// TIA Portal V20 export
TYPE "LCFL_typeMTPMonBinVlv"
TITLE = MTP for monitoring binary valve / MTP für binäre Ventilüberwachung
// MTP data for bistable valve with the feedback monitoring / MTP-Daten für bistabiles Ventil mit Rückmeldeüberwachung
   STRUCT
      WQC { ExternalWritable := 'False'} : Byte := 16#FF;   // Schlechtester Quality Code / Worst quality code
      OSLevel : Byte := 16#00;   // OS-Level / OS level
      StateChannel { ExternalWritable := 'False'} : Bool := FALSE;   // Auswahl des aktiven Betriebsart-Interaktionskanals (0: Die Bedienschalter (*Op) sind zu verwenden; 1: Die automatischen Schalter (*Aut) sind zu verwenden) / Selection of the active operation mode interaction channel (0: The operator switches (*Op) shall be used; 1: The automatic switches (*Aut) shall be used)
      StateOffAut { ExternalWritable := 'False'} : Bool := FALSE;   // Betriebsart durch automatische Interaktion auf "Aus" setzen (relevant, wenn StateChannel = 1) (1: Betriebsart ist auf "Aus" eingestellt; 0: Kein Vorgang) / Set operation mode to "offline" by automatic interaction (relevant, if StateChannel = 1) (1: Operation mode is set to "offline"; 0: No operation)
      StateOpAut { ExternalWritable := 'False'} : Bool := FALSE;   // Betriebsart durch automatische Interaktion auf "Bediener" setzen (relevant, wenn StateChannel = 1) (1: Betriebsart ist auf "Bediener" eingestellt; 0: Kein Vorgang) / Set operation mode to "operator" by automatic interaction (relevant, if StateChannel = 1) (1: Operation mode is set to "manual"; 0: No operation)
      StateAutAut { ExternalWritable := 'False'} : Bool := FALSE;   // Betriebsart durch automatische Interaktion auf "Automatik" setzen (relevant, wenn StateChannel = 1) (1: Betriebsart ist auf "Automatik" eingestellt; 0: Kein Vorgang) / Set operation mode to "automatic" by automatic interaction (relevant, if StateChannel = 1) (1: Operation mode is set to "automatic"; 0: No operation)
      StateOffOp : Bool := FALSE;   // Betriebsart durch Bedienerinteraktion auf "Aus" setzen (relevant, wenn StateChannel = 0) (0-->1: Anforderung, die Betriebsart auf "Aus" zu setzen; 1-->0: Von PEA bestätigen) / Set operation mode to "offline" by operator interaction (relevant, if StateChannel = 0) (0-->1: Request to set operation mode to "offline"; 1-->0: Acknowledge by PEA)
      StateOpOp : Bool := FALSE;   // Betriebsart durch Bedienerinteraktion auf "Bediener" setzen (relevant, wenn StateChannel = 0) (0-->1: Anforderung, die Betriebsart "Bediener" zu setzen; 1-->0: Von PEA bestätigen) / Set operation mode to "operator" by operator interaction (relevant, if StateChannel = 0) (0-->1: Request to set operation mode to "manual"; 1-->0: Acknowledge by PEA)
      StateAutOp : Bool := FALSE;   // Betriebsart durch Bedienerinteraktion auf "Automatik" setzen (relevant, wenn StateChannel = 0) (0-->1: Anforderung, die Betriebsart auf "Automatik" zu setzen; 1-->0: Von PEA bestätigen) / Set operation mode to "automatic" by operator interaction (relevant, if StateChannel = 0) (0-->1: Request to set operation mode is to "automatic"; 1-->0: Acknowledge by PEA)
      StateOpAct { ExternalWritable := 'False'} : Bool := FALSE;   // 1: Aktueller Modus ist "Bediener"; 0: Aktueller Modus ist nicht "Bediener" / 1: Current mode is "operator"; 0: Current mode is not "operator"
      StateAutAct { ExternalWritable := 'False'} : Bool := FALSE;   // 1: Aktueller Modus ist "Automatik"; 0: Aktueller Modus ist nicht "Automatik" / 1: Current mode is "automatic"; 0: Current mode is not "automatic"
      StateOffAct { ExternalWritable := 'False'} : Bool := FALSE;   // 1: Aktueller Modus ist "Aus"; 0: Aktueller Modus ist nicht "Aus" / 1: Current mode is "offline"; 0: Current mode is not "offline"
      SafePos { ExternalWritable := 'False'} : Bool := FALSE;   // Sicherheitsposition (1: Offen; 0: Geschlossen) / Safe position (1: Open; 0: Close)
      SafePosEn { ExternalWritable := 'False'} : Bool := TRUE;   // Hardware-Sicherheitsposition aktiviert (1: Gerät hat eine Sicherheitsposition; 0: Gerät hat keine Sicherheitsposition) / Hardware safe position enabled (1: Device has a safe position; 0: Device has no safe position)
      SafePosAct { ExternalWritable := 'False'} : Bool := FALSE;   // Sicherheitsposition aktiviert (1: Sicherheitsposition ist aktiviert (sicherer Betrieb); 0: Sicherheitsposition ist nicht aktiviert (normaler Betrieb)) / Safe position activated (1: Safe position is activated (safe operation); 0: Safe position is not activated (normal operation))
      OpenOp : Bool := FALSE;   // Öffnen-Befehl von Bediener (relevant, wenn StateOpAct = 1) (0-->1: Anforderung von POL; 1-->0: Bestätigen von PEA) / Open command from operator (relevant, if StateOpAct = 1) (0-->1: Request from POL; 1-->0: Acknowledge from PEA)
      CloseOp : Bool := FALSE;   // Schließen-Befehl von Bediener (relevant, wenn StateOpAct = 1) (0-->1: Request from POL; 1-->0: Acknowledge from PEA) / Close command from operator (relevant, if StateOpAct = 1) (0-->1: Request from POL; 1-->0: Acknowledge from PEA)
      OpenAut { ExternalWritable := 'False'} : Bool := FALSE;   // Ventil auf "Öffnen" von Automatik setzen (relevant, wenn StateAutAct = 1) (1: Anforderung "öffnen"; 0: Anforderung "nicht öffnen") / Set valve to "open" by automatic (relevant, if StateAutAct = 1) (1: Open request; 0: No open request)
      CloseAut { ExternalWritable := 'False'} : Bool := FALSE;   // Ventil auf "Schließen" von Automatik setzen (relevant, wenn StateAutAct = 1) (1: Anforderung "schließen"; 0: Anforderung "nicht schließen") / Set valve to "close" by automatic (relevant, if StateAutAct = 1) (1: Close request; 0: No close request)
      Ctrl { ExternalWritable := 'False'} : Bool := FALSE;   // Ventilsteuerung (1: Gewünschte Position ist "offen"; 0: Gewünschte Position ist "geschlossen") / Valve control (1: Desired position is "open"; 0: Desired position is "closed")
      OpenFbkCalc { ExternalWritable := 'False'} : Bool := FALSE;   // Öffnen-Rückmeldequelle (1: Berechnet; 0: Sensorerkennung) / Open feedback source (1: Calculated; 0: Sensor detection)
      OpenFbk { ExternalWritable := 'False'} : Bool := FALSE;   // Öffnen-Rückmeldesignal (1: Öffnen; 0: Ist nicht geöffnet) / Open feedback signal (1: Open; 0: Is not opened)
      CloseFbkCalc { ExternalWritable := 'False'} : Bool := FALSE;   // Schließen-Rückmeldequelle (1: Berechnet; 0: Sensorerkennung) / Close feedback source (1: Calculated; 0: Sensor detection)
      CloseFbk { ExternalWritable := 'False'} : Bool := FALSE;   // Schließen-Rückmeldesignal (1: Schließen; 0: Ist nicht geschlossen) / Close feedback signal (1: Close; 0: Is not closed)
      PermEn { ExternalWritable := 'False'} : Bool := TRUE;   // Aktiviert die Berechtigungssperre (1: Aktiviert; 0: Deaktiviert) / Enables the permission lock (1: Enabled; 0: Disabled)
      Permit { ExternalWritable := 'False'} : Bool := TRUE;   // Permit erlaubt die Bedienung (1: Berechtigung ist gegeben; 0: Berechtigung ist nicht gegeben) / Permit allows control (1: Permission is given; 0: Permission is not given)
      IntlEn { ExternalWritable := 'False'} : Bool := TRUE;   // Aktiviert die Verriegelungssperre (1: Aktiviert; 0: Deaktiviert) / Enables the interlock lock (1: Enabled; 0: Disabled)
      Interlock { ExternalWritable := 'False'} : Bool := TRUE;   // Interlock verhindert einen Zustandswechsel und bringt das Objekt in die Sicherheitsposition (1: Verriegelung ist nicht aktiv; 0: Verriegelung ist aktiv) / Interlock prevents from being activated and sets object to safe position (1: Interlock is not active; 0: Interlocking is active)
      ProtEn { ExternalWritable := 'False'} : Bool := TRUE;   // Aktiviert die Schutzsperre (1: Aktiviert; 0: Deaktiviert) / Enables the protection lock (1: Enabled; 0: Disabled)
      Protect { ExternalWritable := 'False'} : Bool := TRUE;   // Protect verhindert einen Zustandswechsel und bringt das Objekt in die Sicherheitsposition, ein Zurücksetzen ist erforderlich (1: Schutz ist nicht aktiv; 0: Schutz ist aktiv, erfordert ein Zurücksetzen) / Protect prevents from being activated and sets object to safe position, requires a reset command (1: Protect is not active; 0: Protect is active, requires reset)
      ResetOp : Bool := FALSE;   // Zurücksetzen von Bediener (0-->1: Anforderung von POL; 1-->0: Bestätigen von PEA) / Reset from operator (0-->1: Request from POL; 1-->0: Acknowledge from PEA)
      ResetAut { ExternalWritable := 'False'} : Bool := FALSE;   // Zurücksetzen von Automatik (1: Zurücksetzen ausgeführt; 0: Kein Vorgang) / Reset from automatic (1: Reset executed; 0: No operation)
      MonEn : Bool := TRUE;   // Überwachung aktivieren (1: Aktiviert; 0: Deaktiviert) / Monitor enable (1: Enabled; 0: Disabled)
      MonSafePos { ExternalWritable := 'False'} : Bool := FALSE;   // Fehlerverhalten festlegen, wenn ein Fehler auftritt (1: Nachdem ein Fehler aufgetreten ist, wird die Sicherheitsposition gesetzt; 0: Nachdem ein Fehler aufgetreten ist, hält die Entität den Status) / Set the error behavior, if an error occurs (1: After an error occurs, the safe position will be set; 0: After an error occurs, the entity holds the state)
      MonStatErr { ExternalWritable := 'False'} : Bool := FALSE;   // Statischer Fehler aktiv (1: Aktiv; 0: Inaktiv) / Static error active (1: Active; 0: Inactive)
      MonDynErr { ExternalWritable := 'False'} : Bool := FALSE;   // Dynamischer Fehler aktiv (1: Aktiv; 0: Inaktiv) / Dynamic error active (1: Active; 0: Inactive)
      MonStatTi { ExternalWritable := 'False'} : Real := 0.0;   // Überwachungszeit für ungesteuerte Änderungen [s] / Monitor time for uncontrolled changes [s]
      MonDynTi { ExternalWritable := 'False'} : Real := 0.0;   // Überwachungszeit für gesteuerte Änderungen [s] / Monitor time for controlled changes [s]
   END_STRUCT;
END_TYPE
